FUNCTION F_ITC_SendISR : BOOL
(**************************************************************************************
 * 	Application		:	BoxControl Framework
 *	Revision		:	$Revision: 404529 $
 *	Revision date	:	$Date: 2018-04-23 08:21:38 +0200 (Mo., 23 Apr 2018) $
 *	Last changed by	:	$Author: b7bolm $
 *	URL				:	$URL: http://almscdc.swisslog.com/repo/SWPD/Development/BoxControlFramework/20_Release/trunk/01_Software/BCF/BCF/JumpStart/20_Product/10_App/11_Com/10_Lib/10_Conv/11_ITC/F_ITC_SendISR.TcPOU $
 *
 *	Purpose			:	Wrap message - ISR
 *
 * ------------------------------------------------------------------------------------
 *	Copyright Swisslog [IP AG], Switzerland. All rights reserved.
 * 
 * ------------------------------------------------------------------------------------
 *	
 * 	Revision History: 
 *
 * 	VERSION			DATE			INITIALS			DESCRIPTION
 *	0.1				01.01.2001		swl					Example
 *
 **************************************************************************************)
VAR_INPUT
	eChannelSrc			: E_MFCS_Channel; // Source communicaton channel		
	SignalType			: INT; // Signal Type (0=Inputs, 1=Outputs, 2=Positions)
	StartSignalNumber	: INT; // Start Signal Number
	DataLength			: INT; // Data Length
	Information			: STRING(99); // (HEX) Information Data
	eReturnCode			: E_ErrorConv; // Return code
END_VAR
VAR
	ISR					: ST_ITC_ISR; 
END_VAR

// Map values
ISR.StartSignalNumber := StartSignalNumber;
ISR.SignalType := SignalType;
ISR.DataLength := DataLength;
ISR.Information := Information;
ISR.ReturnCode := eReturnCode;

// Forward to ITC
F_ITC_SendISR := fbITC_Manager.M_SendData(
					meChannel	:= eChannelSrc,
					mMsgType	:= E_ITC_MsgTypeConv.I_O_STATUS_REPORT,
					mpData		:= ADR(ISR),
					mLen		:= SIZEOF(ISR));

END_FUNCTION

(* stored: Version 1.1.0.1, ProductVersion 3.1.4022.12
   POU F_ITC_SendISR: Id {3eb37990-a406-4964-b4f7-deae4b1fa8c4}, SpecialFunc None *)
